FUNCTION_BLOCK FB_DelayAction
VAR_INPUT
END_VAR
VAR_OUTPUT
END_VAR
VAR
	aTimer 		: ARRAY[1..cNoOfTimers] OF TON;
	nTimerNr 	: USINT; 
END_VAR

VAR CONSTANT
	cNoOfTimers : USINT := 4;
END_VAR

FOR nTimerNr := 1 TO cNoOfTimers BY 1 DO
	aTimer[nTimerNr]();
END_FOR

METHOD M_GetProgress : USINT
VAR_INPUT
	nTimerNr	: USINT;
END_VAR

VAR
	nPT : UDINT;
	nET : UDINT;
END_VAR
nPT := TIME_TO_UDINT(aTimer[nTimerNr].PT);
nET := TIME_TO_UDINT(aTimer[nTimerNr].ET);
M_GetProgress := UDINT_TO_USINT(nET * 100 / nPT);
END_METHOD

METHOD M_GetRestTime : TIME
VAR_INPUT
	nTimerNr	: USINT;
END_VAR
IF aTimer[nTimerNr].IN THEN
	M_GetRestTime := aTimer[nTimerNr].PT - aTimer[nTimerNr].ET;
END_IF
END_METHOD

METHOD M_ReleaseAll
VAR_INPUT
END_VAR
FOR nTimerNr := 1 TO cNoOfTimers BY 1 DO
	aTimer[nTimerNr](IN:= FALSE);
END_FOR
END_METHOD

METHOD M_ReleaseTimer
VAR_INPUT
	nTimerNr	: USINT;
END_VAR
aTimer[nTimerNr](IN:= FALSE);
END_METHOD

METHOD M_StartTimer : USINT
VAR_INPUT
	tTime	: TIME;
END_VAR
//nächsten freien Timer suchen
FOR nTimerNr := 1 TO cNoOfTimers BY 1 DO
	IF aTimer[nTimerNr].IN = FALSE THEN
		aTimer[nTimerNr](IN:= TRUE, PT:= tTime);
		M_StartTimer := nTimerNr;
		EXIT;
	END_IF
END_FOR
END_METHOD

END_FUNCTION_BLOCK

(* stored: Version 1.1.0.1, ProductVersion 3.1.4022.10
   POU FB_DelayAction: Id {57afda79-5a94-4310-8123-bd274b19e46d}, SpecialFunc None
   Method M_GetProgress: Id {070a9e0b-d9a4-4ab2-bf39-c8ee27bc7db9}
   Method M_GetRestTime: Id {4b252fea-e37c-42ec-8c0b-9dc7b3252838}
   Method M_ReleaseAll: Id {446e6440-4b0e-4feb-bac7-db1482395ff6}
   Method M_ReleaseTimer: Id {09fb348e-f693-4f14-8ac5-7de201cb47f3}
   Method M_StartTimer: Id {3c1ca161-c9c2-41bc-b7bf-2252dd6f1376} *)
